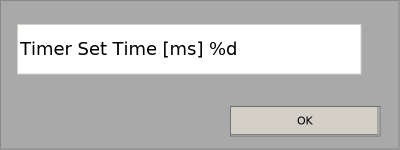
VISUALIZATION DialogTimer_HeaterOn  // 400x150
    Button (230,106 150x30), "OK"
        OnMouseClick: CloseDialog Dialog=DialogTimer_HeaterOn, Result=OK, NumpadKeypadSet=True
    Textfield (17,24 344x50), "Timer Set Time [ms] %d", text variable: PersistentStruct.TimerHotWeldingOn
        OnMouseClick: write the text variable via Edit
END_VISUALIZATION

(* stored: Version 1.1.0.1, ProductVersion 3.1.4024.3
   Visu DialogTimer_HeaterOn: Id {90862752-e15c-467f-8bf6-d6632eefe3aa} *)
